// TwinCAT 3 PLC project RTNNIgen
// Title: Real-Time Neural Network generator
// Company: ISW
// Author: Zexu Zhou, Christoph Hinze
// ProjectVersion: 0.1
// ProgramVersion: 3.1.4024.0
// libraries:
//   Tc2_Standard, * (Beckhoff Automation GmbH)
//   Tc2_System, * (Beckhoff Automation GmbH)
//   Tc3_Module, * (Beckhoff Automation GmbH)
// project tree:
//   DUTs/ act_type.TcDUT, Layer.TcDUT (not stored)
//   / PlcTask.TcTTO (not stored)
//   POUs/ FB_LoadWeights.TcPOU (not stored), F_denormalization.TcPOU (not stored), F_Dot.TcPOU (not stored), F_exponential.TcPOU (not stored), F_ForwardPropagation.TcPOU, F_normalization.TcPOU (not stored), F_relu.TcPOU (not stored), F_selu.TcPOU, F_sigmoid.TcPOU, F_silu.TcPOU, F_softplus.TcPOU, F_softsign.TcPOU (not stored), F_tanh.TcPOU, MAIN.TcPOU
// real-time tasks:
//   TASK PlcTask: cycle T#10ms, priority 20, ADS port 350
//   TASK PlcTask1: cycle T#10ms, priority 21, ADS port 351

// ---- DUTs/act_type.TcDUT
{attribute 'qualified_only'}
{attribute 'strict'}
TYPE act_type :
(
	linear := 0,
	relu :=1,
	tanh :=2,
	sigmoid :=3,
	softplus := 4,
	softsign := 5,
	silu := 6,
	selu := 7,
	exponential := 8,
	normalization := 10,
	denormalization :=11
);
END_TYPE

// ---- POUs/F_ForwardPropagation.TcPOU
FUNCTION F_ForwardPropagation : LREAL
VAR_INPUT
	layer_pre : Layer;
	layer_next : Layer;
	pointer_in : POINTER TO LREAL;
	pointer_out : POINTER TO LREAL; 
END_VAR
VAR
	i : UINT;
	length_in : UINT;	
	length_out : UINT;

	activation_type : act_type;
END_VAR

length_in := layer_pre.num_neurons;
length_out := layer_next.num_neurons;
activation_type := layer_next.activation;
FOR i := 0 TO length_out-1 DO
	pointer_out[i] := F_Dot(ADR(layer_next.pointer_weight[i * length_in]),pointer_in,length_in); 
	pointer_out[i] := layer_next.pointer_bias[i] + pointer_out[i];
	CASE activation_type OF
		act_type.relu:
		pointer_out[i] := F_relu(pointer_out[i]);
		act_type.tanh:
		pointer_out[i] := F_tanh(pointer_out[i]);
		act_type.exponential:
		pointer_out[i] := F_exponential(pointer_out[i]);
		act_type.selu:
		pointer_out[i] := F_selu(pointer_out[i]);
		act_type.sigmoid:
		pointer_out[i] := F_sigmoid(pointer_out[i]);
		act_type.silu:
		pointer_out[i] := F_silu(pointer_out[i]);
		act_type.softplus:
		pointer_out[i] := F_softplus(pointer_out[i]);
		act_type.softsign:
		pointer_out[i] := F_softsign(pointer_out[i]);
	ELSE
		CONTINUE;
	END_CASE
END_FOR

END_FUNCTION

// ---- POUs/F_tanh.TcPOU
FUNCTION F_tanh : LREAL
VAR_INPUT
	x: LREAL;
END_VAR

IF x > 10E6 THEN
	F_tanh := 1;
ELSIF x < -10E6 THEN
	F_tanh := -1;
ELSE
	F_tanh := (EXP(x) - EXP(-x))/(EXP(x) + EXP(-x));
END_IF

END_FUNCTION

// ---- POUs/F_selu.TcPOU
FUNCTION F_selu : lreal
VAR_INPUT
	x : LREAL;
END_VAR
VAR
	scale : LREAL := 1.05070098;
	alpha : LREAL := 1.67326324;
END_VAR

IF x > 0 THEN
	F_selu := scale * x;
ELSE
	F_selu := scale * alpha * (exp(x) - 1);
END_IF

END_FUNCTION

// ---- POUs/F_sigmoid.TcPOU
FUNCTION F_sigmoid : LREAL
VAR_INPUT
	x : LREAL;
END_VAR

F_sigmoid := 1 / (1 + exp(-x));

END_FUNCTION

// ---- POUs/F_silu.TcPOU
FUNCTION F_silu : lreal
VAR_INPUT
	x : LREAL;
END_VAR

F_silu := x / (1 + exp(-x));

END_FUNCTION

// ---- POUs/F_softplus.TcPOU
FUNCTION F_softplus : lreal
VAR_INPUT
	x : LREAL;
END_VAR

F_softplus := log(exp(x)+1);

END_FUNCTION

// ---- POUs/MAIN.TcPOU
PROGRAM MAIN
VAR
END_VAR

END_PROGRAM
